FUNCTION_BLOCK PtInterval IMPLEMENTS I_PtInterval
VAR_INPUT
END_VAR
VAR_OUTPUT
END_VAR
VAR
	_Start : PtDateTime;
	_End : PtDateTime;
	_Absolute : BOOL;
	
	_DeltaYears : DINT;
	_DeltaMonths : DINT;
	_DeltaDays : DINT;
END_VAR

PROPERTY Absolute : BOOL
GET
Absolute := _Absolute;
END_GET
SET
_Absolute := Absolute;
END_SET
END_PROPERTY

PROPERTY End : PtDateTime
GET
End := _End;
END_GET
SET
_End := End;
END_SET
END_PROPERTY

METHOD inMonth : DINT
VAR_INPUT
END_VAR
inMonth := ABS(_Start.Month - _End.Month);
END_METHOD

METHOD inYears : DINT
VAR_INPUT
END_VAR
inYears := ABS(_Start.Year - _End.Year);
END_METHOD

METHOD Set //: BOOL
VAR_INPUT
	Start : PtDateTime;
	End : PtDateTime;
	Absolute : BOOL;
END_VAR
_Start := Start;
_End := End;
_Absolute := Absolute;

_DeltaYears := ABS(_Start.Year - _End.Year);
_DeltaMonths := ABS(_Start.Month - _End.Month);
_DeltaDays := ABS(_Start.Day - End.Day);
END_METHOD

PROPERTY Start : PtDateTime
GET
END_GET
SET
_Start := Start;
END_SET
END_PROPERTY

END_FUNCTION_BLOCK

(* stored: Version 1.1.0.1, ProductVersion 3.1.4024.12
   POU PtInterval: Id {81e6146b-efef-4ffa-9681-6b446ef612b5}, SpecialFunc None
   Property Absolute: Id {850a2711-42a4-4649-beeb-ad46908d4db0}
   Get Get: Id {84ffecba-217a-467b-ba14-629eaf1ac184}
   Set Set: Id {8fb06fe2-f8c9-4026-b802-0d19fabefb26}
   Property End: Id {49b7ccff-456b-497f-a7b9-d266cbdbd9ff}
   Get Get: Id {c51f9c78-b544-41ec-9f9d-93c674039eae}
   Set Set: Id {8fb38c71-0620-4cad-8753-041ac8d238bf}
   Method inMonth: Id {9d54fa83-e390-4b1d-8489-8dd5ccaf61df}
   Method inYears: Id {929b505f-fdb0-4a02-b5bd-122a78ebd708}
   Method Set: Id {ad7ecb83-8faa-4b59-b16c-52d8de52e79d}
   Property Start: Id {dcdc2291-7714-4af6-b419-dadfb6c86870}
   Get Get: Id {cda418ee-7804-4d2c-9d18-68fad9af9a9d}
   Set Set: Id {32da7c98-855d-41f4-87a4-60baa0d6b62c} *)
